FUNCTION ifExprFunc1: BOOL
VAR_INPUT
    dummy: INT;
END_VAR

IF (func_f1(farg_f1_p:=TRUE)) THEN
    ifExprFunc1 := TRUE;
ELSE
    ifExprFunc1 := TRUE;
END_IF;

END_FUNCTION

(* stored: ProductVersion 3.1.0.18, Version 1.1.0.1 *)
